{attribute 'GeneratedUsingTerminal: EL3413-0000-0016'}
{attribute addProperty BoxType "EL3413-0000-0016"}
{attribute addProperty Id "IndexAT %Q*USINT1ChannelAT %Q*USINT1"}
{attribute addProperty CRC "1807848559"}
{attribute addProperty Size "2"}
TYPE PM_Outputs_Auxiliary_6BC1946F EXTENDS OutputBase_10CEE7DE :
STRUCT
	{attribute addProperty Name "Index"}
	Index AT %Q* : USINT;
	{attribute addProperty Name "Channel"}
	Channel AT %Q* : USINT;
END_STRUCT
END_TYPE

(* stored: Version 1.2.0.0, ProductVersion 3.1.4024.9
   DUT PM_Outputs_Auxiliary_6BC1946F: Id {5a08e2b7-4178-46b6-b654-896fd5d8439c} *)
